(*
SPDX-FileCopyrightText: © 2026 Oleksandr Tiutyk <trofimich@gmail.com>
SPDX-License-Identifier: MIT
License: https://opensource.org/license/mit
*)

(*!
<summary>Defines a composite activity that executes at most one active child activity at a time.</summary>
*)

INTERFACE IExclusiveCompositeActivity EXTENDS ICompositeActivity

(*!
<summary>Returns the currently selected child activity, or 0 when no child is selected.</summary>
*)
{attribute 'monitoring' := 'call'}
PROPERTY CurrentActivity : IActivity
GET
END_GET
END_PROPERTY

END_INTERFACE

(* stored: Version 1.1.0.1
   Itf IExclusiveCompositeActivity: Id {eb197991-df55-4e73-a57a-6882e69e164f}
   Property CurrentActivity: Id {ae9ff0e6-470a-4b29-9027-1c30fa80b4e4}
   Get Get: Id {748e4b23-96d2-4b60-a68a-28dd4e3ce9cf} *)
